PROGRAM PRG_Compilation
VAR
	senStart				: FB_Sensor_NO;
    senEnd					: FB_Sensor_NO;
    evActuator				: FB_Electrovalve_5on2_1Coil;

	fbActuator				: FB_Actuator (
								senStart	:= senStart,
	                            senEnd		:= senEnd,
	                            evControl	:= evActuator
							);	
END_VAR

END_PROGRAM

(* stored: Version 1.1.0.1
   POU PRG_Compilation: Id {d24d79c3-2ef5-49a9-88ed-c4ba78e1268d}, SpecialFunc None *)
